PROGRAM PRG_PMPS
VAR
    fbArbiterIO : FB_SubSysToArbiter_IO;
END_VAR

g_FastFaultOutputK0.Execute(
	i_xVeto:=PMPS_GVL.stCurrentBeamParameters.aStoppers[PMPS.K_Stopper.MR1K1_IN] OR PMPS_GVL.stCurrentBeamParameters.aStoppers[PMPS.K_Stopper.MR1K3_IN], 
	bAutoReset:=TRUE
);

// Aggregate FastFaultOutputs into a single FastFault
g_FastFault(
	io_fbFFHWO := g_FastFaultOutputAll,
	i_xOK := (  g_FastFaultOutputK0.q_xFastFaultOut 
				AND g_FastFaultOutputK0.q_xFastFaultOut
				AND g_FastFaultOutputK2.q_xFastFaultOut
				AND g_FastFaultOutputK3.q_xFastFaultOut
				AND g_FastFaultOutputK4.q_xFastFaultOut
			 )
);
// Arbiter
fbArbiterIO(Arbiter := g_fbArbiter1, fbFFHWO := g_FastFaultOutputK0);

END_PROGRAM

(* stored: Version 1.1.0.1, ProductVersion 3.1.4024.2
   POU PRG_PMPS: Id {f7d360c9-1fd6-4e06-b31d-7f5233ed9ceb}, SpecialFunc None *)
